// TIA Portal V17 export
// export: Created 2025-03-10T13:12:10.3840547Z, ExportSetting WithDefaults, DisplayName Totally Integrated Automation Portal, DisplayVersion V17 Update 8, DisplayName TIA Portal Openness, DisplayVersion V17 Update 8, DisplayName TIA Portal Version Control Interface, DisplayVersion V17, DisplayName SINAMICS Startdrive Advanced, DisplayVersion V17 SP2, DisplayName SINAMICS Startdrive G110M, G120, G120C, G120D, G120P, G115D, DisplayVersion V17 SP2, DisplayName SINAMICS Startdrive G130, G150, S120, S150, SINAMICS MV, S210, DisplayVersion V17 SP2, DisplayName STEP 7 Professional, DisplayVersion V17 Update 8, DisplayName SINUMERIK ONE STEP 7 Toolbox, DisplayVersion V17 Update 12, DisplayName SINUMERIK 840D sl STEP 7 Toolbox, DisplayVersion V17 Update 12, DisplayName STEP 7 Safety, DisplayVersion V17 Update 6, DisplayName WinCC Advanced, DisplayVersion V17 Update 8
TYPE "ASPIRATION"
// stored: IsFailsafeCompliant false
   STRUCT
      GENERAL_CONDITIONS : Bool;   // GENERAL CONDITIONS
      SWITCH_ON_CONDITIONS : Bool;   // ADVANCE CONDITIONS / SWITCH ON CONDITIONS
      SWITCH_OFF_CONDITIONS : Bool;   // RETURN CONDITIONS / SWITCH OFF CONDITIONS
      GENERAL_CONDITIONS_HELP : Bool;   // GENERAL CONDITIONS HELP
      SWITCH_ON_CONDITIONS_HELP : Bool;   // SWITCH ON CONDITIONS HELP
      SWITCH_OFF_CONDITIONS_HELP : Bool;   // SWITCH OFF CONDITIONS HELP
      SWITCH_ON_HMI_REQUEST : Bool;   // ADVANCE HMI REQUEST / SWITCH ON MANUAL HMI REQUEST
      SWITCH_OFF_HMI_REQUEST : Bool;   // RETURN HMI REQUEST / SWITCH OFF MANUAL HMI REQUEST
      SWITCH_ON_MANUAL_REQUEST : Bool;   // ADVANCE MANUAL REQUEST / SWITCH ON MANUAL REQUEST
      SWITCH_OFF_MANUAL_REQUEST : Bool;   // RETURN MANUAL REQUEST / SWITCH OFF MANUAL REQUEST
      SWITCH_ON_AUTO_REQUEST : Bool;   // ADVANCE AUTO REQUEST / SWITCH ON AUTO REQUEST
      SWITCH_OFF_AUTO_REQUEST : Bool;   // RETURN AUTO REQUEST / SWITCH OFF AUTO REQUEST
      SWITCH_ON_GLOBAL_REQUEST : Bool;   // ADVANCE GLOBAL REQUEST / SWITCH ON GLOBAL REQUEST
      SWITCH_OFF_GLOBAL_REQUEST : Bool;   // RETURN GLOBAL REQUEST / SWITCH OFF GLOBAL REQUEST
      SWITCH_ON_COMMAND : Bool;   // ADVANCE COMMAND / SWITCH ON COMMAND
      SWITCH_OFF_COMMAND : Bool;   // RETURN COMMAND / SWITCH OFF COMMAND
      FULL_SWITCHED_ON : Bool;   // ADVANCED FEEDBACK / SWITCHED ON AND COMMANDED
      FULL_SWITCHED_OFF : Bool;   // RETURNED FEEDBACK / SWITCHED OFF AND COMMANDED
      SIMULTANEITY_ALARM : Bool;   // SIMULTANEITY FAULT / SIMULTANEITY ALARM
      TIME_EXCEEDED_ALARM : Bool;   // TIME EXCEEDED / TIME EXCEEDED ALARM
      ANY_ACTIVE_ALARM : Bool;   // FAULT / ANY ACTIVE ALARM
      IS_SEOC_ALARMS : Bool;   // INMEDIATE STOP AND STOP END OF CYCLE ALARMS
      PULSE_1 : Bool;   // PULSE 1
      PULSE_2 : Bool;   // PULSE 2
      PULSE_3 : Bool;   // PULSE 3
   END_STRUCT;
END_TYPE
